# EPICS autosave request: iocBoot/iocMARCCD/auto_settings.req
file "ADBase_settings.req",       P=$(P),  R=cam1:
file "marCCD_settings.req",       P=$(P),  R=cam1:
file "NDFile_settings.req",       P=$(P),  R=cam1:
file "NDPluginBase_settings.req", P=$(P),  R=image1:
file "NDStdArrays_settings.req",  P=$(P),  R=image1:
file "NDPluginBase_settings.req", P=$(P),  R=ROI1:
file "NDROI_settings.req",        P=$(P),  R=ROI1:
file "NDROIN_settings.req",       P=$(P),  R=ROI1:0:
file "NDROIN_settings.req",       P=$(P),  R=ROI1:1:
file "NDROIN_settings.req",       P=$(P),  R=ROI1:2:
file "NDROIN_settings.req",       P=$(P),  R=ROI1:3:
file "scan_settings.req",         P=$(P)cam1: S=scan1
file "scan_settings.req",         P=$(P)cam1: S=scan2
file "scan_settings.req",         P=$(P)cam1: S=scan3
file "scan_settings.req",         P=$(P)cam1: S=scan4
